// TIA Portal project "Tetsi" (V15.1)

(* hardware
DEVICE "S71500/ET200MP station_1"  S7-1500 station
   slot 0: "Rail_0"  Rack  6ES7 590-1***0-0AA0
   slot 1: "PLC_1"  CPU 1511-1 PN  6ES7 511-1AK02-0AB0  V2.6
      slot 3: "CPU display_1"  6ES7591-1AA00-0AA0
   slot 2: "DI 16x24VDC / DQ 16x24VDC/0.5A BA_1"  DI 16/DQ 16x24VDC  6ES7 523-1BL00-0AA0  V1.0
   slot 3: "AI/AQ 4xU/I/RTD/TC / 2xU/I ST_1"  AI/AQ 4xU/I/RTD/TC / 2xU/I ST  6ES7 534-7QE00-0AB0  V1.0
*)

// ===== PLC "PLC_1"  CPU 1511-1 PN =====

VAR_GLOBAL   // PLC tag table "Default tag table"
   "Clock_Byte" AT %MB0 : Byte;
   "Clock_10Hz" AT %M0.0 : Bool;
   "Clock_5Hz" AT %M0.1 : Bool;
   "Clock_2.5Hz" AT %M0.2 : Bool;
   "Clock_2Hz" AT %M0.3 : Bool;
   "Clock_1.25Hz" AT %M0.4 : Bool;
   "Clock_1Hz" AT %M0.5 : Bool;
   "Clock_0.625Hz" AT %M0.6 : Bool;
   "Clock_0.5Hz" AT %M0.7 : Bool;
   "Tag_3" AT %M8.0 : Bool;
   "Tag_1" AT %M8.1 : Bool;
   "Tag_4" AT %Q0.2 : Bool;
END_VAR

VAR_GLOBAL   // PLC tag table "Tagit"
   "start" AT %M10.0 : Bool;
   "stop" AT %M10.1 : Bool;
   "anturi1" AT %M10.2 : Bool;
   "anturi2" AT %M10.3 : Bool;
   "turvakytkin" AT %M10.4 : Bool;
   "moottori1" AT %Q0.0 : Bool;
   "moottori2" AT %Q0.1 : Bool;
   "aktuaattori" AT %M10.6 : Bool;
   "akt_max" AT %M10.7 : Bool;
   "akt_min" AT %M11.0 : Bool;
   "actBtn" AT %M11.1 : Bool;
END_VAR

DATA_BLOCK "DB"   // DB1
{ S7_Optimized_Access := 'FALSE' }
VERSION : 0.1
   VAR
      nLaatikoita : Int;
   END_VAR
BEGIN
END_DATA_BLOCK

DATA_BLOCK "Data_block_1"   // DB2
{ S7_Optimized_Access := 'FALSE' }
VERSION : 0.1
   VAR
      start : Bool;
      stop : Bool;
      anturi1 : Bool;
      turvakytkin : Bool;
      moottori1 : Bool;
   END_VAR
BEGIN
END_DATA_BLOCK

ORGANIZATION_BLOCK "Main"   // OB1, LAD, ProgramCycle
TITLE = "Main Program Sweep (Cycle)"
{ S7_Optimized_Access := 'TRUE' }
VERSION : 0.1
   VAR_INPUT
      Initial_Call : Bool;   // Initial call of this OB
      Remanence : Bool;   // =True, if remanent data are available
   END_VAR
   VAR_TEMP   // added for the SCL form of the ladder/FBD networks
      _w1 : Bool;
   END_VAR
BEGIN

REGION Network 1
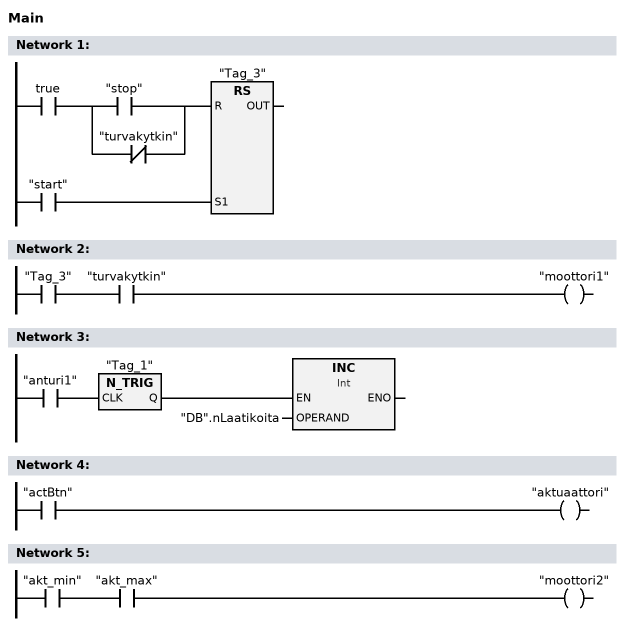
   RUNG wire#powerrail
      Contact( true )
      wire#w1
      Contact( "stop" )
      wire#w2
      S_RS(operand := "Tag_3", s1 := wire#w3)
   END_RUNG
   RUNG wire#w1
      I_Contact( "turvakytkin" )
   END_RUNG wire#w2
   RUNG wire#powerrail
      Contact( "start" )
   END_RUNG wire#w3
   // the same network as SCL:
   IF true AND ("stop" OR NOT "turvakytkin") THEN
       "Tag_3" := FALSE;   // RS flip-flop
   END_IF;
   IF "start" THEN "Tag_3" := TRUE; END_IF;
END_REGION

REGION Network 2
   RUNG wire#powerrail
      Contact( "Tag_3" )
      Contact( "turvakytkin" )
      Coil( "moottori1" )
   END_RUNG
   // the same network as SCL:
   "moottori1" := "Tag_3" AND "turvakytkin";
END_REGION

REGION Network 3
   RUNG wire#powerrail
      Contact( "anturi1" )
      N_Trig( "Tag_1" )
      { S7_Templates := "DestType := Int" } Inc( "DB".nLaatikoita )
   END_RUNG
   // the same network as SCL:
   #_w1 := NOT "anturi1" AND "Tag_1";   // falling edge
   "Tag_1" := "anturi1";
   IF #_w1 THEN "DB".nLaatikoita := "DB".nLaatikoita + 1; END_IF;
END_REGION

REGION Network 4
   RUNG wire#powerrail
      Contact( "actBtn" )
      Coil( "aktuaattori" )
   END_RUNG
   // the same network as SCL:
   "aktuaattori" := "actBtn";
END_REGION

REGION Network 5
   RUNG wire#powerrail
      Contact( "akt_min" )
      Contact( "akt_max" )
      Coil( "moottori2" )
   END_RUNG
   // the same network as SCL:
   "moottori2" := "akt_min" AND "akt_max";
END_REGION
END_ORGANIZATION_BLOCK